Universal Robots PolyScope program: wrs2020_taskboard_retainer_and_nut.urp

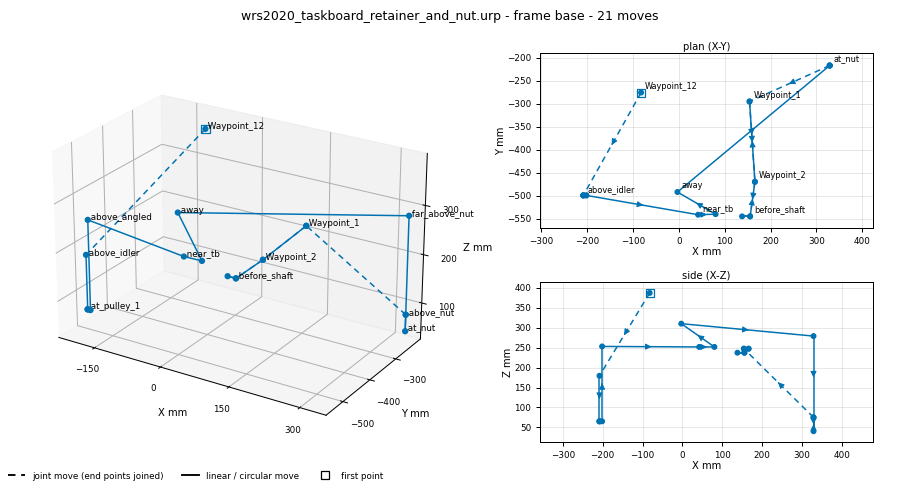
[picture p0: tool path of wrs2020_taskboard_retainer_and_nut.urp in frame base, 21 of 21 moves have a stored position in this frame; points joined in program order, loops and branches not executed]
Program wrs2020_taskboard_retainer_and_nut (installation=default directory=/programs createdIn=5.6.0.90886 lastSavedIn=5.6.0.90886 robotSerialNumber=20205500180)
Calibrated DH parameters: a=[0.000135, -0.030981, -0.334292, 0.000083, 0.000088, 0]; d=[0.162656, 258.79096, -331.603246, 72.945842, 0.099724, 0.099562]; alpha=[1.569535, 0.001639, 0.002824, 1.569633, -1.569323, 0]; deltaTheta=[0, 1.497881, -2.049261, 0.551379, 0, 0]
Robot Program (runOnlyOnce=true)
  MoveJ speed 60 deg/s, acceleration 80 deg/s^2 (useActiveTCP=true) feature=Base
    Waypoint Waypoint_12: TCP in base x=-82.102 y=-275.549 z=387.348 mm, rx=-0.1814 ry=-3.1114 rz=0.2863 rad; joints [35.849, -127.007, 98.51, -68.6, -82.206, -47.132] deg; TCP offset x=0 y=0 z=220 mm, rx=0 ry=0 rz=0 rad
  URCap Gripper (Robotiq_Grippers, Robotiq Inc.) dataModel(position=44.705882352941174, force=100.0, speed=100.0, positionInDouble=44.705882352941174, forceInDouble=100.0, speedInDouble=100.0, slaveIds=[9], blocking=true)
  MoveJ speed 60 deg/s, acceleration 80 deg/s^2 (useActiveTCP=true) feature=Base
    Waypoint above_idler: TCP in base x=-208.011 y=-499.592 z=179.536 mm, rx=2.2188 ry=-2.2117 rz=-0.0634 rad; joints [54.601, -83.96, 96.653, -102.683, -92.188, -125.564] deg
  MoveL speed 50 mm/s, acceleration 1200 mm/s^2 (useActiveTCP=true) feature=Base
    Waypoint at_pulley_1: motionParameters(jointSpeed=1.047198 jointAcceleration=1.396263 cartesianSpeed=0.5 cartesianAcceleration=1.2); TCP in base x=-208.011 y=-499.592 z=65.293 mm, rx=2.2188 ry=-2.2117 rz=-0.0634 rad; joints [54.588, -78.262, 107.874, -119.601, -92.18, -125.521] deg
  URCap Gripper (Robotiq_Grippers, Robotiq Inc.) dataModel(position=100.0, force=0.0, speed=0.0, positionInDouble=100.0, forceInDouble=0.0, speedInDouble=0.0, slaveIds=[9], blocking=true)
  URCap Gripper (Robotiq_Grippers, Robotiq Inc.) dataModel(position=44.705882352941174, force=100.0, speed=100.0, positionInDouble=44.705882352941174, forceInDouble=100.0, speedInDouble=100.0, slaveIds=[9], blocking=true)
  MoveL speed 50 mm/s, acceleration 1200 mm/s^2 (useActiveTCP=true) feature=Base
    Waypoint at_pulley_2: motionParameters(jointSpeed=1.047198 jointAcceleration=1.396263 cartesianSpeed=0.5 cartesianAcceleration=1.2); TCP in base x=-208.002 y=-499.584 z=65.278 mm, rx=-0.0091 ry=-3.107 rz=-0.0353 rad; joints [54.587, -78.261, 107.874, -119.597, -92.178, -35] deg
  URCap Gripper (Robotiq_Grippers, Robotiq Inc.) dataModel(position=100.0, force=0.0, speed=0.0, positionInDouble=100.0, forceInDouble=0.0, speedInDouble=0.0, slaveIds=[9], blocking=true)
  URCap Gripper (Robotiq_Grippers, Robotiq Inc.) dataModel(position=57.64705882352941, force=100.0, speed=100.0, positionInDouble=57.64705882352941, forceInDouble=100.0, speedInDouble=100.0, slaveIds=[9], blocking=true)
  MoveL speed 50 mm/s, acceleration 1200 mm/s^2 (useActiveTCP=true) feature=Base
    Waypoint at_pulley_1: motionParameters(jointSpeed=1.047198 jointAcceleration=1.396263 cartesianSpeed=0.5 cartesianAcceleration=1.2); TCP in base x=-208.011 y=-499.592 z=65.293 mm, rx=2.2188 ry=-2.2117 rz=-0.0634 rad; joints [54.588, -78.262, 107.874, -119.601, -92.18, -125.521] deg
  MoveL speed 50 mm/s, acceleration 1200 mm/s^2 (useActiveTCP=true) feature=Base
    Waypoint angled: motionParameters(jointSpeed=1.047198 jointAcceleration=1.396263 cartesianSpeed=0.5 cartesianAcceleration=1.2); TCP in base x=-201.431 y=-499.592 z=65.293 mm, rx=1.8379 ry=-1.8459 rz=-0.6644 rad; joints [74.44, -74.851, 119.325, -144.728, -127.06, -108.593] deg
  URCap Gripper (Robotiq_Grippers, Robotiq Inc.) dataModel(position=100.0, force=0.0, speed=0.0, positionInDouble=100.0, forceInDouble=0.0, speedInDouble=0.0, slaveIds=[9], blocking=true)
  MoveL speed 50 mm/s, acceleration 1200 mm/s^2 (useActiveTCP=true) feature=Base
    Waypoint above_angled: TCP in base x=-201.431 y=-499.592 z=253.175 mm, rx=1.8379 ry=-1.8459 rz=-0.6644 rad; joints [74.47, -88.384, 103.414, -115.34, -127.048, -108.685] deg
  MoveL speed 250 mm/s, acceleration 1200 mm/s^2 (useActiveTCP=true) feature=Base
    Waypoint near_tb: TCP in base x=42.161 y=-541.658 z=251.88 mm, rx=-2.2078 ry=1.5258 rz=-1.5075 rad; joints [47.035, -95.124, 115.286, -91.003, -33.11, -164.164] deg
    Waypoint in_ridge: motionParameters(jointSpeed=1.047198 jointAcceleration=1.396263 cartesianSpeed=0.02 cartesianAcceleration=1.2); TCP in base x=80.326 y=-540.51 z=251.883 mm, rx=-2.2141 ry=1.5067 rz=-1.5032 rad; joints [50.981, -96.869, 118.023, -96.662, -32.219, -158.618] deg
  Popup Message (haltProgram=false message=wait for screw tool to hold inputType=Text)
  URCap Gripper (Robotiq_Grippers, Robotiq Inc.) dataModel(position=41.96078431372549, force=100.0, speed=100.0, positionInDouble=41.96078431372549, forceInDouble=100.0, speedInDouble=100.0, slaveIds=[9], blocking=true)
  MoveL speed 250 mm/s, acceleration 1200 mm/s^2 (useActiveTCP=true) feature=Base
    Waypoint away: TCP in base x=-2.896 y=-492.237 z=310.294 mm, rx=-2.2141 ry=1.5067 rz=-1.5032 rad; joints [37.989, -98.984, 106.815, -66.013, -37.422, -179.666] deg
    Waypoint far_above_nut: TCP in base x=328.886 y=-216.609 z=279.114 mm, rx=1.7144 ry=1.9308 rz=0.7284 rad; joints [87.485, -126.161, 121.652, -76.577, -49.859, -282.701] deg
  MoveL speed 250 mm/s, acceleration 1200 mm/s^2 (useActiveTCP=true) feature=Base
    Waypoint above_nut: TCP in base x=328.886 y=-216.609 z=75.372 mm, rx=1.7144 ry=1.9308 rz=0.7284 rad; joints [87.428, -116.788, 148.991, -113.328, -49.811, -282.641] deg
    URCap Gripper (Robotiq_Grippers, Robotiq Inc.) dataModel(position=67.84313725490196, force=100.0, speed=100.0, positionInDouble=67.84313725490196, forceInDouble=100.0, speedInDouble=100.0, slaveIds=[9], blocking=true)
    Waypoint at_nut: TCP in base x=328.886 y=-216.609 z=40.536 mm, rx=1.7144 ry=1.9308 rz=0.7284 rad; joints [87.407, -110.975, 152.75, -122.912, -49.807, -282.622] deg
    URCap Gripper (Robotiq_Grippers, Robotiq Inc.) dataModel(position=100.0, force=0.0, speed=0.0, positionInDouble=100.0, forceInDouble=0.0, speedInDouble=0.0, slaveIds=[9], blocking=true)
    Waypoint above_nut: TCP in base x=328.886 y=-216.609 z=75.372 mm, rx=1.7144 ry=1.9308 rz=0.7284 rad; joints [87.428, -116.788, 148.991, -113.328, -49.811, -282.641] deg
  MoveJ speed 60 deg/s, acceleration 80 deg/s^2 (useActiveTCP=true) feature=Base
    Waypoint Waypoint_1: TCP in base x=154.205 y=-294.953 z=247.483 mm, rx=-1.9267 ry=-2.1381 rz=0.3655 rad; joints [112.572, -107.181, 108.526, -84.751, -108.754, -252.336] deg
    Waypoint Waypoint_2: TCP in base x=165.947 y=-469.896 z=247.483 mm, rx=-1.8555 ry=-2.0623 rz=0.4684 rad; joints [110.013, -83.157, 88.588, -87.029, -115.402, -254.126] deg
    Waypoint before_shaft: TCP in base x=155.498 y=-545.232 z=237.455 mm, rx=-1.6624 ry=-1.781 rz=0.723 rad; joints [114.093, -65.084, 72.827, -73.388, -131.867, -240.378] deg
  MoveL speed 250 mm/s, acceleration 1200 mm/s^2 (useActiveTCP=true) feature=Base
    Waypoint at_shaft: TCP in base x=138.013 y=-545.232 z=237.455 mm, rx=-1.6624 ry=-1.781 rz=0.723 rad; joints [112.688, -66.576, 75.262, -75.498, -132.428, -242.113] deg
    Popup Message (haltProgram=false message=wait for screw tool to hold inputType=Text)
    URCap Gripper (Robotiq_Grippers, Robotiq Inc.) dataModel(position=67.84313725490196, force=100.0, speed=100.0, positionInDouble=67.84313725490196, forceInDouble=100.0, speedInDouble=100.0, slaveIds=[9], blocking=true)
    Waypoint before_shaft: TCP in base x=155.498 y=-545.232 z=237.455 mm, rx=-1.6624 ry=-1.781 rz=0.723 rad; joints [114.093, -65.084, 72.827, -73.388, -131.867, -240.378] deg
    Waypoint Waypoint_2: TCP in base x=165.947 y=-469.896 z=247.483 mm, rx=-1.8555 ry=-2.0623 rz=0.4684 rad; joints [110.013, -83.157, 88.588, -87.029, -115.402, -254.126] deg
    Waypoint Waypoint_1: TCP in base x=154.205 y=-294.953 z=247.483 mm, rx=-1.9267 ry=-2.1381 rz=0.3655 rad; joints [112.572, -107.181, 108.526, -84.751, -108.754, -252.336] deg
